FUNCTION_BLOCK FB_Xbox_1D_Joystick_NC
VAR
	_mcJog				: MC_Jog;
	_mcHalt				: MC_Halt;
	_rtJogEnable		: R_TRIG;
	_ftJogEnable		: F_TRIG;
	_bJoggingActive		: BOOL;
	_fPrevOverride		: UDINT;
END_VAR

METHOD FB_init : BOOL
VAR_INPUT
	bInitRetains : BOOL; // if TRUE, the retain variables are initialized (warm start / cold start)
	bInCopyCode : BOOL;  // if TRUE, the instance afterwards gets moved into the copy code (online change)
END_VAR
END_METHOD

METHOD Jog
VAR_INPUT
	bEnable			: BOOL;	
	fJoystick		: LREAL;
	Axis			: REFERENCE TO Axis_Ref;
	stOptions		: ST_Xbox_1D_Joystick_NC_Options;
END_VAR
VAR
	bJogForward 	: BOOL;
	bJogBackwards 	: BOOL;
END_VAR
// Rising edge trigger of the block enable
_rtJogEnable(CLK := bEnable);
// Falling edge trigger of the block enable
_ftJogEnable(CLK := bEnable);

// Halt the axis in case of Enable falling off
_mcHalt(Axis		 := Axis, 
		Execute		 := _ftJogEnable.Q,
    	Deceleration := stOptions.stXbox_NC_Halt_Dynamics.fDeceleration, 
   		Jerk         := stOptions.stXbox_NC_Halt_Dynamics.fJerk,
		BufferMode	 := stOptions.stXbox_NC_Halt_Dynamics.mcBufferMode,
		Options		 := stOptions.stXbox_NC_Halt_Dynamics.stOptions);

// Rising edge trigger of the block enable
IF _rtJogEnable.Q THEN
	// Save the current override value before jogging
	// Check the Axis reference is valid	
	IF __ISVALIDREF(Axis) THEN
		THIS^._fPrevOverride := Axis.PlcToNc.Override;
	END_IF
	// Enable the jog methods
	_bJoggingActive	:= TRUE;
END_IF

// Falling edge trigger of the block enable
IF _ftJogEnable.Q THEN
	// Restore the past override value before enable
	// Check the Axis reference is valid	
	IF __ISVALIDREF(Axis) THEN
		Axis.PlcToNc.Override := THIS^._fPrevOverride;
			// Cleanup any old Jog commands
		THIS^._mcJog(
					  Axis:= Axis, 
					  JogForward:= FALSE, 
					  JogBackwards:= FALSE, 
					  Mode:= E_JogMode.MC_JOGMODE_STANDARD_FAST);	
	END_IF
	// Disable calling to jog methods
	_bJoggingActive := FALSE;
END_IF

// Check the Joystick reference is valid
IF _bJoggingActive THEN
	// Check the Axis reference is valid	
	IF __ISVALIDREF(Axis) THEN
		// Check the direction the joystick is moving, or if in deadzone					 
		IF fJoystick = 0 THEN
			bJogForward 	:= FALSE;
			bJogBackwards := FALSE;
			Axis.PlcToNc.Override := 0;
		ELSIF fJoystick < 0 THEN
			// Check for inversion
			IF NOT stOptions.bInverted THEN
				bJogForward 	:= FALSE;
				bJogBackwards := TRUE;
			ELSE
				bJogForward 	:= TRUE;
				bJogBackwards := FALSE;
			END_IF
			// Set the new override based on the directional pressure
			Axis.PlcToNc.Override := TO_UDINT(ABS(fJoystick * (stOptions.fMaxOverride/100)) * 10000);
		ELSIF fJoystick > 0 THEN
			// Check for inversion
			IF NOT stOptions.bInverted THEN
				bJogForward 	:= TRUE;
				bJogBackwards := FALSE;
			ELSE
				bJogForward 	:= FALSE;
				bJogBackwards := TRUE;
			END_IF
			// Set the new override based on the directional pressure
			Axis.PlcToNc.Override := TO_UDINT(ABS(fJoystick * (stOptions.fMaxOverride/100)) * 10000);
		END_IF
		// Main jog call for axis
		THIS^._mcJog(
					  Axis:= Axis, 
					  JogForward:= bJogForward, 
					  JogBackwards:= bJogBackwards, 
					  Mode:= E_JogMode.MC_JOGMODE_STANDARD_FAST);
	END_IF
END_IF
END_METHOD

END_FUNCTION_BLOCK

(* stored: Version 1.1.0.1, ProductVersion 3.1.4024.11
   POU FB_Xbox_1D_Joystick_NC: Id {2ba681f7-602b-4d57-80a3-58d7cfe103fa}, SpecialFunc None
   Method FB_init: Id {0aa70316-42f0-49a2-8556-e9aebc66a94b}
   Method Jog: Id {9a4b5f71-5b33-4177-bb28-505a96ce8cf6} *)
